FUNCTION_BLOCK GET_STRUCT_VALUE (* Service Interface Function Block Type *)
  PACKAGE eclipse4diac::convert;
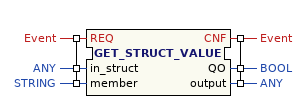
  EVENT_INPUT
    REQ WITH member, in_struct; (* Get Value out of structure *)
  END_EVENT
  EVENT_OUTPUT
    CNF WITH QO, output; (* REQ event finished *)
  END_EVENT
  VAR_INPUT
    in_struct : ANY; (* Structure to look into *)
    member : STRING; (* Member of the strucuture to retrieve. Inner members are access using the dot (.) operator *)
  END_VAR
  VAR_OUTPUT
    QO : BOOL; (* TRUE if no errors ocurred, FALSE otherwise *)
    output : ANY; (* Selected member if QO = TRUE, remains unchanged otherwise *)
  END_VAR
END_FUNCTION_BLOCK
